{attribute 'qualified_only'}
VAR_GLOBAL CONSTANT
	// Encoder reference values in counts = nm
	// Enc Ref Vals from alignment 2020-6-12
	nYUP_ENC_REF : ULINT := 13611000;
	nYDWN_ENC_REF : ULINT := 13433600;
	nXUP_ENC_REF : ULINT := 25210500;
	nXDWN_ENC_REF : ULINT := 24971800;
END_VAR

(* stored: Version 1.1.0.1, ProductVersion 3.1.4022.18
   GVL GVL_MR1L4_Constants: Id {bab5a8a7-7e61-4255-b9b1-a7508819eb64} *)
